FUNCTION_BLOCK FeedReactor3PsBasic (* Logica das 3 bombas de alimentacao (2 servico + 1 reserva) - mesmo funcionamento da Water Discharge *)
  (* Standard: 61499-2 *)
  (* Version 1.2, 10/7/2026, Claude/Hidryco, Schneider Electric, Rev3 - Velocidade das bombas sempre igual a saida do PID (1 ou 2 bombas); so muda para C2 na entrada/troca de bomba; sem fator 2, sem Cmin e sem capacidade teorica na falha do medidor | Rev2 - Setpoint do PID sempre igual ao setpoint do Nereda (removida a troca pela vazao medida com as bombas em C2) | Rev1 - Reescrito conforme a narrativa (cap. 2) com o mesmo funcionamento da Water Discharge (Rev13): Cmax/C2/C3/Cmin em % de velocidade; entrada da 2a com a bomba no Cmax pela velocidade real (narrativa); descida ate C2 confirmada pela velocidade real antes de partir a nova; T_C2 com as bombas em C2; reserva em falha parte na hora em C2; saida da 2a com protecao anti-ciclo; rodizio por horimetro; paradas por LL do buffer, pH/condutividade (L/H, retomada apos T_Restart) e vazao LL (T_FlowLL, retomada apos T_Restart); falha do medidor pela capacidade teorica; status para IHM *)
  PACKAGE SE.Nereda;
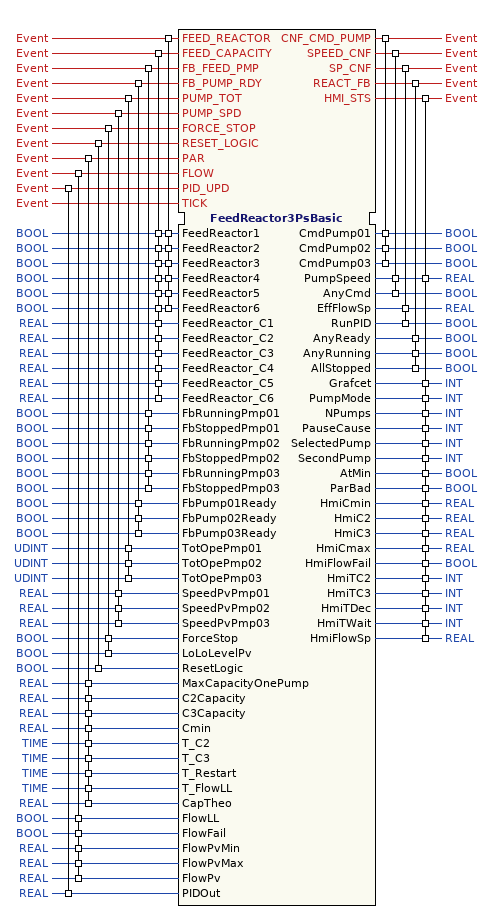
  EVENT_INPUT
    FEED_REACTOR WITH FeedReactor1, FeedReactor2, FeedReactor3, FeedReactor4, FeedReactor5, FeedReactor6; (* Pedido de alimentacao dos reatores (StartFeeding) *)
    FEED_CAPACITY WITH FeedReactor1, FeedReactor2, FeedReactor3, FeedReactor4, FeedReactor5, FeedReactor6, FeedReactor_C1, FeedReactor_C2, FeedReactor_C3, FeedReactor_C4, FeedReactor_C5, FeedReactor_C6; (* Setpoint de vazao dos reatores [m3/h] *)
    FB_FEED_PMP WITH FbRunningPmp01, FbStoppedPmp01, FbRunningPmp02, FbStoppedPmp02, FbRunningPmp03, FbStoppedPmp03;
    FB_PUMP_RDY WITH FbPump01Ready, FbPump02Ready, FbPump03Ready;
    PUMP_TOT WITH TotOpePmp01, TotOpePmp02, TotOpePmp03; (* Horimetro das bombas (rodizio) *)
    PUMP_SPD WITH SpeedPvPmp01, SpeedPvPmp02, SpeedPvPmp03; (* Velocidade real das bombas [%] *)
    FORCE_STOP WITH ForceStop, LoLoLevelPv; (* LL do buffer (40LT0001) e pH/condutividade fora da faixa (L/H) *)
    RESET_LOGIC WITH ResetLogic;
    PAR WITH MaxCapacityOnePump, C2Capacity, C3Capacity, Cmin, T_C2, T_C3, T_Restart, T_FlowLL, CapTheo; (* Parametros *)
    FLOW WITH FlowLL, FlowFail, FlowPvMin, FlowPvMax, FlowPv; (* Status e valor do 40FT0003 *)
    PID_UPD WITH PIDOut; (* Saida do PID *)
    TICK; (* Base de tempo 1 s *)
  END_EVENT
  EVENT_OUTPUT
    CNF_CMD_PUMP WITH CmdPump01, CmdPump02, CmdPump03; (* Comando das bombas *)
    SPEED_CNF WITH PumpSpeed, AnyCmd; (* Velocidade enviada a cada bomba em servico *)
    SP_CNF WITH EffFlowSp, RunPID; (* Setpoint efetivo e liberacao do PID *)
    REACT_FB WITH AnyReady, AnyRunning, AllStopped; (* Retorno das bombas para os reatores *)
    HMI_STS WITH Grafcet, PumpMode, NPumps, PauseCause, SelectedPump, SecondPump, PumpSpeed, AtMin, ParBad, HmiCmin, HmiC2, HmiC3, HmiCmax, HmiFlowFail, HmiTC2, HmiTC3, HmiTDec, HmiTWait, HmiFlowSp; (* Status para a IHM (a cada 1 s e na mudanca) *)
  END_EVENT
  VAR_INPUT
    FeedReactor1 : BOOL; (* StartFeeding do reator 1 (fase Feed em RUN e AV41101 aberta) *)
    FeedReactor2 : BOOL; (* StartFeeding do reator 2 (fase Feed em RUN e AV41101 aberta) *)
    FeedReactor3 : BOOL; (* StartFeeding do reator 3 (fase Feed em RUN e AV41101 aberta) *)
    FeedReactor4 : BOOL; (* StartFeeding do reator 4 (fase Feed em RUN e AV41101 aberta) *)
    FeedReactor5 : BOOL; (* StartFeeding do reator 5 (fase Feed em RUN e AV41101 aberta) *)
    FeedReactor6 : BOOL; (* StartFeeding do reator 6 (fase Feed em RUN e AV41101 aberta) *)
    FeedReactor_C1 : REAL; (* Setpoint de vazao do reator 1 [m3/h] *)
    FeedReactor_C2 : REAL; (* Setpoint de vazao do reator 2 [m3/h] *)
    FeedReactor_C3 : REAL; (* Setpoint de vazao do reator 3 [m3/h] *)
    FeedReactor_C4 : REAL; (* Setpoint de vazao do reator 4 [m3/h] *)
    FeedReactor_C5 : REAL; (* Setpoint de vazao do reator 5 [m3/h] *)
    FeedReactor_C6 : REAL; (* Setpoint de vazao do reator 6 [m3/h] *)
    FbRunningPmp01 : BOOL;
    FbStoppedPmp01 : BOOL;
    FbRunningPmp02 : BOOL;
    FbStoppedPmp02 : BOOL;
    FbRunningPmp03 : BOOL;
    FbStoppedPmp03 : BOOL;
    FbPump01Ready : BOOL;
    FbPump02Ready : BOOL;
    FbPump03Ready : BOOL;
    TotOpePmp01 : UDINT; (* Horimetro da bomba 1 *)
    TotOpePmp02 : UDINT; (* Horimetro da bomba 2 *)
    TotOpePmp03 : UDINT; (* Horimetro da bomba 3 *)
    SpeedPvPmp01 : REAL; (* Velocidade real da bomba 1 [%] *)
    SpeedPvPmp02 : REAL; (* Velocidade real da bomba 2 [%] *)
    SpeedPvPmp03 : REAL; (* Velocidade real da bomba 3 [%] *)
    ForceStop : BOOL; (* pH ou condutividade fora da faixa (alarmes L/H dos analisadores) *)
    LoLoLevelPv : BOOL; (* Nivel LL do buffer 40LT0001 *)
    ResetLogic : BOOL; (* Nao usado (compatibilidade) *)
    MaxCapacityOnePump : REAL; (* Cmax: velocidade de 1 bomba acima da qual entra a 2a [%] *)
    C2Capacity : REAL; (* C2: velocidade das bombas na entrada de uma nova bomba [%] *)
    C3Capacity : REAL; (* C3: velocidade das 2 bombas abaixo da qual sai 1 [%] *)
    Cmin : REAL; (* Nao atua desde a Rev3 (velocidade minima = OutMin do PID); so exibido na IHM *)
    T_C2 : TIME; (* Tempo com as bombas em C2 *)
    T_C3 : TIME; (* Tempo abaixo de C3 *)
    T_Restart : TIME; (* Tempo de espera para retomar a alimentacao (pH/condutividade/vazao LL) *)
    T_FlowLL : TIME; (* Vazao LL do 40FT0003 com bomba rodando por este tempo = para a alimentacao (0 = desabilitado) *)
    CapTheo : REAL; (* Nao usada desde a Rev3 (na falha do medidor as bombas seguem a saida do PID) *)
    FlowLL : BOOL; (* Alarme LL do 40FT0003 *)
    FlowFail : BOOL; (* Falha do 40FT0003 *)
    FlowPvMin : REAL; (* Inicio de faixa do 40FT0003 *)
    FlowPvMax : REAL; (* Fim de faixa do 40FT0003 *)
    FlowPv : REAL; (* Vazao medida 40FT0003 [m3/h] (nao usada desde a Rev2; mantida pela ligacao no FeedReactorLogic) *)
    PIDOut : REAL; (* Saida do PID = velocidade de cada bomba em servico [%] *)
  END_VAR
  VAR_OUTPUT
    CmdPump01 : BOOL;
    CmdPump02 : BOOL;
    CmdPump03 : BOOL;
    PumpSpeed : REAL; (* Velocidade enviada a cada bomba em servico [%] (= saida do PID; C2 na entrada/troca de bomba) *)
    AnyCmd : BOOL; (* Alguma bomba comandada *)
    EffFlowSp : REAL; (* Setpoint do PID [m3/h] = setpoint do Nereda (maior pedido entre os reatores alimentando) *)
    RunPID : BOOL; (* PID em automatico *)
    AnyReady : BOOL; (* Alguma bomba disponivel (Ready ou rodando) *)
    AnyRunning : BOOL; (* Alguma bomba rodando *)
    AllStopped : BOOL; (* Nenhuma bomba rodando *)
    Grafcet : INT; (* 0 sem pedido | 3 alimentando *)
    PumpMode : INT; (* 0=1 bomba 1=reduzindo p/ C2 2=nova bomba em C2 (T_C2) 3=duas no PID *)
    NPumps : INT; (* Bombas em servico rodando *)
    PauseCause : INT; (* 0 sem pausa | 1 nivel LL 40LT0001 | 2 pH/condutividade | 3 vazao LL 40FT0003 *)
    SelectedPump : INT; (* Bomba em servico ha mais tempo *)
    SecondPump : INT; (* Segunda bomba em servico *)
    AtMin : BOOL; (* Sempre FALSE desde a Rev3 (sem velocidade minima na logica) *)
    ParBad : BOOL; (* Parametros incoerentes (so aviso) *)
    HmiCmin : REAL;
    HmiC2 : REAL;
    HmiC3 : REAL;
    HmiCmax : REAL;
    HmiFlowFail : BOOL;
    HmiTC2 : INT; (* Tempo em C2 [s] *)
    HmiTC3 : INT; (* Tempo abaixo de C3 [s] *)
    HmiTDec : INT; (* Tempo descendo ate C2 [s] *)
    HmiTWait : INT; (* Tempo de espera para retomar [s] *)
    HmiFlowSp : REAL; (* Setpoint de vazao [m3/h] *)
  END_VAR
  VAR
    Paused : BOOL;
    FeedReq : BOOL;
    FlowSp : REAL;
    Dem : REAL;
    CminEff : REAL;
    C2Eff : REAL;
    SpdRaw : REAL;
    ParOk : BOOL;
    ExitCond : BOOL;
    Spare : BOOL;
    SpdAtC2 : BOOL;
    SpdUpC2 : BOOL;
    SpdAtMax : BOOL;
    NCmd : INT;
    NRun : INT;
    NWant : INT;
    PumpSel : INT;
    MinTot : UDINT;
    MinOrd : UDINT;
    Seq : UDINT;
    Ord1 : UDINT;
    Ord2 : UDINT;
    Ord3 : UDINT;
    Tacc : TIME;
    T3acc : TIME;
    Tdec : TIME;
    Tup : TIME;
    Trest : TIME;
    Tmax : TIME;
    Tll : TIME;
    TC2s : INT;
    TC3s : INT;
    TDecs : INT;
    TRests : INT;
    FromTick : BOOL;
    EdgeOut : BOOL;
    EdgeSpd : BOOL;
    EdgeSts : BOOL;
    EdgeCmd : BOOL;
    PrevSP : REAL;
    PrevRun : BOOL;
    PrevAR : BOOL;
    PrevARun : BOOL;
    PrevSpd : REAL;
    PrevAC : BOOL;
    PrevC1 : BOOL;
    PrevC2 : BOOL;
    PrevC3 : BOOL;
    PrevSPM : INT;
    PrevSNP : INT;
    PrevSPC : INT;
    PrevSGR : INT;
    PrevSAM : BOOL;
    PrevSPB : BOOL;
    TolC2 : REAL := 2.0; (* Parametro interno: tolerancia [%] para considerar a bomba em C2 *)
    T_DecMax : TIME := T#1m; (* Parametro interno: tempo maximo esperando a velocidade real chegar a C2 *)
    HystExit : REAL := 10.0; (* Parametro interno: margem [%] abaixo de Cmax para a bomba que fica apos a saida da 2a (anti-ciclo) *)
  END_VAR
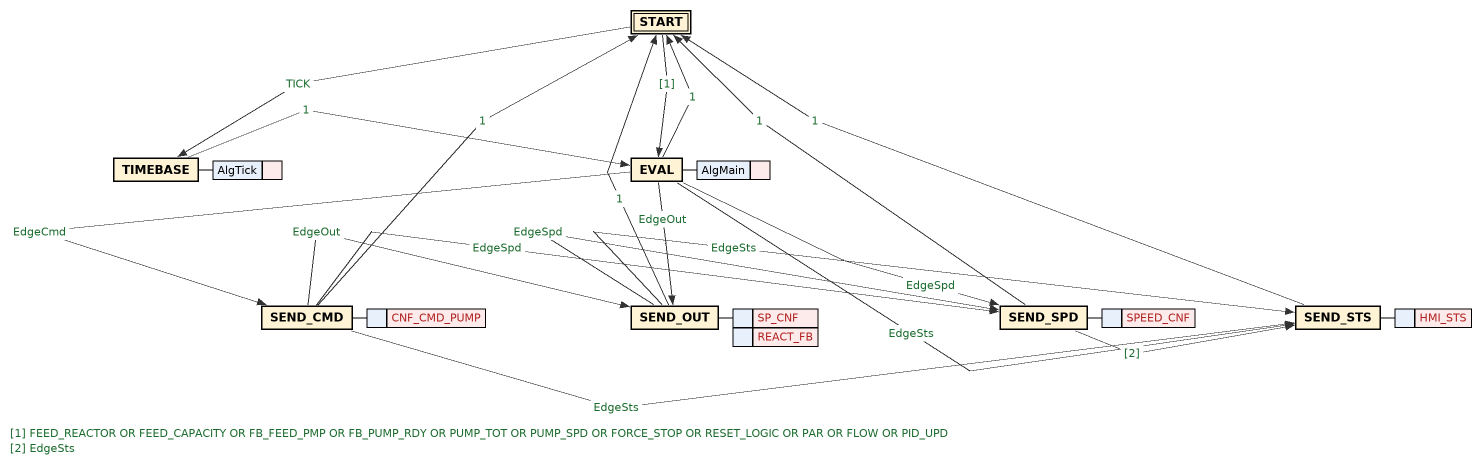
  EC_STATES
    START;
    TIMEBASE : AlgTick;
    EVAL : AlgMain;
    SEND_CMD : -> CNF_CMD_PUMP;
    SEND_OUT : -> SP_CNF, -> REACT_FB;
    SEND_SPD : -> SPEED_CNF;
    SEND_STS : -> HMI_STS;
  END_STATES
  EC_TRANSITIONS
    START TO TIMEBASE := TICK;
    START TO EVAL := FEED_REACTOR OR FEED_CAPACITY OR FB_FEED_PMP OR FB_PUMP_RDY OR PUMP_TOT OR PUMP_SPD OR FORCE_STOP OR RESET_LOGIC OR PAR OR FLOW OR PID_UPD;
    EVAL TO SEND_CMD := EdgeCmd;
    EVAL TO SEND_OUT := EdgeOut;
    EVAL TO SEND_SPD := EdgeSpd;
    EVAL TO SEND_STS := EdgeSts;
    EVAL TO START := 1;
    SEND_CMD TO SEND_OUT := EdgeOut;
    SEND_CMD TO SEND_SPD := EdgeSpd;
    SEND_CMD TO SEND_STS := EdgeSts;
    SEND_CMD TO START := 1;
    SEND_OUT TO SEND_SPD := EdgeSpd;
    SEND_OUT TO SEND_STS := EdgeSts;
    SEND_OUT TO START := 1;
    SEND_SPD TO SEND_STS := EdgeSts;
    SEND_SPD TO START := 1;
    SEND_STS TO START := 1;
    TIMEBASE TO EVAL := 1;
  END_TRANSITIONS
  ALGORITHM AlgMain IN ST: (* Logica das bombas de alimentacao *)
;
(* ============================================================
   FeedReactor3PsBasic Rev3 - bombas de alimentacao P4001/P4002/P4003 (2 servico + 1 reserva)
   Rev3: a velocidade das bombas e SEMPRE a saida do PID (1 ou 2 bombas). So muda para C2 na entrada/troca de bomba
         (modos 1 e 2). Sem fator 2 com uma bomba, sem velocidade minima (Cmin) e sem capacidade teorica na falha do medidor.
   Rev2: o setpoint do PID e sempre o setpoint do Nereda (removida a troca pela vazao medida com as bombas em C2).
   Narrativa cap. 2 (Influent feed) com o mesmo funcionamento da Water Discharge do Sludge Buffer.
   - Partida: StartFeeding de algum reator (fase Feed em RUN e AV41101 aberta). SP = maior pedido [m3/h].
   - Velocidade de cada bomba em servico = saida do PID [%]. Cmax / C2 / C3 em % de velocidade de UMA bomba.
     Limites de velocidade: OutMin/OutMax do proprio PID.
   - Entrada: velocidade REAL da bomba em operacao no Cmax -> a(s) em operacao descem ate C2 (velocidade REAL),
     a nova parte em C2, T_C2 com as duas com velocidade REAL em C2, depois PID. Sem liberacao por tempo.
   - Saida: velocidade REAL de todas as bombas em operacao abaixo de C3 por T_C3: sai a que partiu primeiro.
   - Falha de bomba com 2 em servico: reserva parte na hora, todas em C2, T_C2, depois PID.
   - Paradas: 1 nivel LL 40LT0001 (retoma ao sair o LL) | 2 pH/condutividade fora da faixa (retoma T_Restart apos voltar)
              3 vazao LL 40FT0003 por T_FlowLL com bomba rodando (retoma apos T_Restart)
   - Falha do 40FT0003 (40FT05): as bombas continuam seguindo a saida do PID (Rev3).
   PumpMode: 0 uma bomba | 1 reduzindo p/ C2 (nova parada) | 2 nova em C2 (T_C2) | 3 duas no PID
   ============================================================ *)

(* ---------- 1. Pedido de alimentacao e setpoint ---------- *)
FeedReq := FeedReactor1 OR FeedReactor2 OR FeedReactor3 OR FeedReactor4 OR FeedReactor5 OR FeedReactor6;
FlowSp := 0.0;
IF FeedReactor1 AND (FeedReactor_C1 > FlowSp) THEN
    FlowSp := FeedReactor_C1;
END_IF;
IF FeedReactor2 AND (FeedReactor_C2 > FlowSp) THEN
    FlowSp := FeedReactor_C2;
END_IF;
IF FeedReactor3 AND (FeedReactor_C3 > FlowSp) THEN
    FlowSp := FeedReactor_C3;
END_IF;
IF FeedReactor4 AND (FeedReactor_C4 > FlowSp) THEN
    FlowSp := FeedReactor_C4;
END_IF;
IF FeedReactor5 AND (FeedReactor_C5 > FlowSp) THEN
    FlowSp := FeedReactor_C5;
END_IF;
IF FeedReactor6 AND (FeedReactor_C6 > FlowSp) THEN
    FlowSp := FeedReactor_C6;
END_IF;
IF FeedReq THEN
    Grafcet := 3;
ELSE
    Grafcet := 0;
END_IF;

(* ---------- 2. Demanda e parametros ---------- *)
(* Rev3: a demanda e sempre a saida do PID (inclusive com o medidor em falha) *)
Dem := PIDOut;
IF Dem > 100.0 THEN
    Dem := 100.0;
END_IF;
IF Dem < 0.0 THEN
    Dem := 0.0;
END_IF;
CminEff := Cmin;
IF CminEff > 100.0 THEN
    CminEff := 100.0;
END_IF;
IF CminEff < 0.0 THEN
    CminEff := 0.0;
END_IF;
(* so Cmax e C2 sao indispensaveis; o resto apenas avisa (ParBad) - a protecao anti-ciclo esta embutida na saida *)
ParOk := (MaxCapacityOnePump > 0.0) AND (C2Capacity > 0.0);
(* Rev3: Cmin nao atua mais (velocidade minima = OutMin do PID); 2 x C3 >= Cmax continua causando ciclo de entrada/saida *)
ParBad := (MaxCapacityOnePump <= 0.0) OR (C2Capacity <= 0.0) OR ((2.0 * C3Capacity) >= MaxCapacityOnePump);
C2Eff := C2Capacity;
ExitCond := FALSE; (* calculado mais abaixo, so pela velocidade real das bombas *)

(* ---------- 3. Paradas da alimentacao (narrativa 2.2) ---------- *)
IF Grafcet = 3 THEN
    IF Paused THEN
        IF (PauseCause = 1) AND (NOT LoLoLevelPv) THEN
            Paused := FALSE;
            PauseCause := 0;
            Tll := T#0s;
        ELSIF (PauseCause >= 2) AND (NOT LoLoLevelPv) AND (NOT ForceStop) AND (Trest >= T_Restart) THEN
            Paused := FALSE;
            PauseCause := 0;
            Tll := T#0s;
        END_IF;
    END_IF;
    IF LoLoLevelPv THEN
        Paused := TRUE;
        PauseCause := 1;
        Trest := T#0s;
        TRests := 0;
    ELSIF ForceStop THEN
        Paused := TRUE;
        PauseCause := 2;
        Trest := T#0s;
        TRests := 0;
    ELSIF (NOT Paused) AND (T_FlowLL > T#0s) AND (Tll >= T_FlowLL) THEN
        Paused := TRUE;
        PauseCause := 3;
        Trest := T#0s;
        TRests := 0;
        Tll := T#0s;
    END_IF;
END_IF;

(* ---------- 4. Bombas ---------- *)
IF (Grafcet = 3) AND Paused THEN
    CmdPump01 := FALSE;
    CmdPump02 := FALSE;
    CmdPump03 := FALSE;
    PumpMode := 0;
    Tacc := T#0s;
    TC2s := 0;
    T3acc := T#0s;
    TC3s := 0;
    NCmd := 0;
    NRun := 0;
    EffFlowSp := FlowSp;
    PumpSpeed := 0.0;
    AtMin := FALSE;
ELSIF Grafcet = 3 THEN
    (* 4.1 bomba sai de servico somente se nao estiver Ready (modo programa) NEM Running *)
    IF CmdPump01 AND NOT FbPump01Ready AND NOT FbRunningPmp01 THEN
        CmdPump01 := FALSE;
    END_IF;
    IF CmdPump02 AND NOT FbPump02Ready AND NOT FbRunningPmp02 THEN
        CmdPump02 := FALSE;
    END_IF;
    IF CmdPump03 AND NOT FbPump03Ready AND NOT FbRunningPmp03 THEN
        CmdPump03 := FALSE;
    END_IF;
    NCmd := 0;
    IF CmdPump01 THEN
        NCmd := NCmd + 1;
    END_IF;
    IF CmdPump02 THEN
        NCmd := NCmd + 1;
    END_IF;
    IF CmdPump03 THEN
        NCmd := NCmd + 1;
    END_IF;
    NRun := 0;
    IF CmdPump01 AND FbRunningPmp01 THEN
        NRun := NRun + 1;
    END_IF;
    IF CmdPump02 AND FbRunningPmp02 THEN
        NRun := NRun + 1;
    END_IF;
    IF CmdPump03 AND FbRunningPmp03 THEN
        NRun := NRun + 1;
    END_IF;
    Spare := (FbPump01Ready AND NOT CmdPump01) OR (FbPump02Ready AND NOT CmdPump02) OR (FbPump03Ready AND NOT CmdPump03);
    (* bombas em operacao ja desceram ate C2 (velocidade real) *)
    SpdAtC2 := TRUE;
    IF CmdPump01 AND FbRunningPmp01 AND (SpeedPvPmp01 > (C2Eff + TolC2)) THEN
        SpdAtC2 := FALSE;
    END_IF;
    IF CmdPump02 AND FbRunningPmp02 AND (SpeedPvPmp02 > (C2Eff + TolC2)) THEN
        SpdAtC2 := FALSE;
    END_IF;
    IF CmdPump03 AND FbRunningPmp03 AND (SpeedPvPmp03 > (C2Eff + TolC2)) THEN
        SpdAtC2 := FALSE;
    END_IF;
    (* bomba em operacao com velocidade real ja no Cmax *)
    SpdAtMax := FALSE;
    IF CmdPump01 AND FbRunningPmp01 AND (SpeedPvPmp01 >= (MaxCapacityOnePump - TolC2)) THEN
        SpdAtMax := TRUE;
    END_IF;
    IF CmdPump02 AND FbRunningPmp02 AND (SpeedPvPmp02 >= (MaxCapacityOnePump - TolC2)) THEN
        SpdAtMax := TRUE;
    END_IF;
    IF CmdPump03 AND FbRunningPmp03 AND (SpeedPvPmp03 >= (MaxCapacityOnePump - TolC2)) THEN
        SpdAtMax := TRUE;
    END_IF;
    (* bombas em operacao com velocidade real ja em C2 (subida da que entrou) *)
    SpdUpC2 := TRUE;
    IF CmdPump01 AND FbRunningPmp01 AND (SpeedPvPmp01 < (C2Eff - TolC2)) THEN
        SpdUpC2 := FALSE;
    END_IF;
    IF CmdPump02 AND FbRunningPmp02 AND (SpeedPvPmp02 < (C2Eff - TolC2)) THEN
        SpdUpC2 := FALSE;
    END_IF;
    IF CmdPump03 AND FbRunningPmp03 AND (SpeedPvPmp03 < (C2Eff - TolC2)) THEN
        SpdUpC2 := FALSE;
    END_IF;
    (* saida de uma bomba: velocidade real de TODAS as bombas em operacao abaixo de C3 (sem usar a saida do PID) *)
    ExitCond := NRun >= 2;
    IF CmdPump01 AND FbRunningPmp01 AND (SpeedPvPmp01 >= C3Capacity) THEN
        ExitCond := FALSE;
    END_IF;
    IF CmdPump02 AND FbRunningPmp02 AND (SpeedPvPmp02 >= C3Capacity) THEN
        ExitCond := FALSE;
    END_IF;
    IF CmdPump03 AND FbRunningPmp03 AND (SpeedPvPmp03 >= C3Capacity) THEN
        ExitCond := FALSE;
    END_IF;
    (* 4.1b com 2 bombas (modo 2/3) uma saiu de servico: a reserva parte NA HORA, todas em C2, T_C2, depois PID *)
    IF ParOk AND (PumpMode >= 2) AND (NCmd < 2) THEN
        IF Spare AND (NCmd >= 1) THEN
            PumpMode := 2;
            Tacc := T#0s;
            TC2s := 0;
            Tup := T#0s;
        ELSE
            PumpMode := 0;
        END_IF;
    END_IF;

    (* 4.2 numero de bombas *)
    IF NOT ParOk THEN
        PumpMode := 0;
    ELSIF PumpMode = 0 THEN
        (* entra a 2a bomba somente quando a velocidade REAL da bomba em operacao chega ao Cmax *)
        IF Spare AND (NRun >= 1) AND SpdAtMax THEN
            PumpMode := 1;
            Tdec := T#0s;
            TDecs := 0;
        END_IF;
    ELSIF PumpMode = 1 THEN
        (* a nova so parte depois que a velocidade REAL da(s) bomba(s) em operacao desceu ate C2 *)
        IF (NOT Spare) OR (NCmd = 0) THEN
            PumpMode := 0;
        ELSIF SpdAtC2 THEN
            PumpMode := 2;
            Tacc := T#0s;
            TC2s := 0;
            Tup := T#0s;
        END_IF;
    ELSIF PumpMode = 2 THEN
        (* T_C2 conta com as duas rodando e com velocidade REAL em C2 *)
        IF (NRun >= 2) AND (Tacc >= T_C2) THEN
            PumpMode := 3;
            T3acc := T#0s;
            TC3s := 0;
        END_IF;
    ELSIF PumpMode = 3 THEN
        (* saida: velocidade REAL das bombas abaixo de C3 por T_C3 *)
        IF ExitCond AND (T3acc >= T_C3) THEN
            PumpMode := 0;
            T3acc := T#0s;
            TC3s := 0;
        END_IF;
    END_IF;
    IF PumpMode >= 2 THEN
        NWant := 2;
    ELSE
        NWant := 1;
    END_IF;

    (* 4.3 entra bomba disponivel de menor horimetro (rodizio) - ate 2 vezes *)
    IF NCmd < NWant THEN
        PumpSel := 0;
        IF FbPump01Ready AND NOT CmdPump01 THEN
            PumpSel := 1;
            MinTot := TotOpePmp01;
        END_IF;
        IF FbPump02Ready AND NOT CmdPump02 THEN
            IF (PumpSel = 0) OR (TotOpePmp02 < MinTot) THEN
                PumpSel := 2;
                MinTot := TotOpePmp02;
            END_IF;
        END_IF;
        IF FbPump03Ready AND NOT CmdPump03 THEN
            IF (PumpSel = 0) OR (TotOpePmp03 < MinTot) THEN
                PumpSel := 3;
                MinTot := TotOpePmp03;
            END_IF;
        END_IF;
        IF PumpSel = 1 THEN
            CmdPump01 := TRUE;
            Seq := Seq + 1;
            Ord1 := Seq;
            NCmd := NCmd + 1;
        ELSIF PumpSel = 2 THEN
            CmdPump02 := TRUE;
            Seq := Seq + 1;
            Ord2 := Seq;
            NCmd := NCmd + 1;
        ELSIF PumpSel = 3 THEN
            CmdPump03 := TRUE;
            Seq := Seq + 1;
            Ord3 := Seq;
            NCmd := NCmd + 1;
        END_IF;
    END_IF;
    IF NCmd < NWant THEN
        PumpSel := 0;
        IF FbPump01Ready AND NOT CmdPump01 THEN
            PumpSel := 1;
            MinTot := TotOpePmp01;
        END_IF;
        IF FbPump02Ready AND NOT CmdPump02 THEN
            IF (PumpSel = 0) OR (TotOpePmp02 < MinTot) THEN
                PumpSel := 2;
                MinTot := TotOpePmp02;
            END_IF;
        END_IF;
        IF FbPump03Ready AND NOT CmdPump03 THEN
            IF (PumpSel = 0) OR (TotOpePmp03 < MinTot) THEN
                PumpSel := 3;
                MinTot := TotOpePmp03;
            END_IF;
        END_IF;
        IF PumpSel = 1 THEN
            CmdPump01 := TRUE;
            Seq := Seq + 1;
            Ord1 := Seq;
            NCmd := NCmd + 1;
        ELSIF PumpSel = 2 THEN
            CmdPump02 := TRUE;
            Seq := Seq + 1;
            Ord2 := Seq;
            NCmd := NCmd + 1;
        ELSIF PumpSel = 3 THEN
            CmdPump03 := TRUE;
            Seq := Seq + 1;
            Ord3 := Seq;
            NCmd := NCmd + 1;
        END_IF;
    END_IF;

    (* 4.4 excedente: sai a bomba em operacao ha mais tempo (menor ordem de partida) *)
    IF NCmd > NWant THEN
        PumpSel := 0;
        IF CmdPump01 THEN
            PumpSel := 1;
            MinOrd := Ord1;
        END_IF;
        IF CmdPump02 THEN
            IF (PumpSel = 0) OR (Ord2 < MinOrd) THEN
                PumpSel := 2;
                MinOrd := Ord2;
            END_IF;
        END_IF;
        IF CmdPump03 THEN
            IF (PumpSel = 0) OR (Ord3 < MinOrd) THEN
                PumpSel := 3;
                MinOrd := Ord3;
            END_IF;
        END_IF;
        IF PumpSel = 1 THEN
            CmdPump01 := FALSE;
        ELSIF PumpSel = 2 THEN
            CmdPump02 := FALSE;
        ELSIF PumpSel = 3 THEN
            CmdPump03 := FALSE;
        END_IF;
        NCmd := NCmd - 1;
    END_IF;

    (* 4.5 sem bomba para a 2a posicao: volta a operar com uma *)
    IF (PumpMode >= 2) AND (NCmd < 2) THEN
        PumpMode := 0;
    END_IF;

    (* 4.6 setpoint do PID e velocidade das bombas *)
    (* setpoint do PID = setpoint do Nereda (maior pedido), sempre - nunca trocado pela vazao medida (Rev2) *)
    EffFlowSp := FlowSp;
    (* Rev3: velocidade de cada bomba = saida do PID; a unica sobreposicao e C2 na entrada/troca de bomba (modos 1 e 2) *)
    IF (PumpMode = 1) OR (PumpMode = 2) THEN
        SpdRaw := C2Eff;
    ELSE
        SpdRaw := Dem;
    END_IF;
    IF SpdRaw > 100.0 THEN
        SpdRaw := 100.0;
    END_IF;
    IF SpdRaw < 0.0 THEN
        SpdRaw := 0.0;
    END_IF;
    AtMin := FALSE; (* Rev3: sem velocidade minima na logica *)
    PumpSpeed := SpdRaw;
ELSE
    (* sem pedido de alimentacao *)
    CmdPump01 := FALSE;
    CmdPump02 := FALSE;
    CmdPump03 := FALSE;
    PumpMode := 0;
    Tacc := T#0s;
    TC2s := 0;
    T3acc := T#0s;
    TC3s := 0;
    NCmd := 0;
    NRun := 0;
    EffFlowSp := FlowSp;
    PumpSpeed := 0.0;
    AtMin := FALSE;
    Paused := FALSE;
    PauseCause := 0;
    Trest := T#0s;
    TRests := 0;
    Tll := T#0s;
END_IF;

(* ---------- 5. Saidas ---------- *)
AnyCmd := CmdPump01 OR CmdPump02 OR CmdPump03;
RunPID := (Grafcet = 3) AND (NOT Paused) AND AnyCmd;
AnyReady := FbPump01Ready OR FbRunningPmp01 OR FbPump02Ready OR FbRunningPmp02 OR FbPump03Ready OR FbRunningPmp03;
AnyRunning := FbRunningPmp01 OR FbRunningPmp02 OR FbRunningPmp03;
AllStopped := NOT AnyRunning;
NPumps := NRun;
SelectedPump := 0;
SecondPump := 0;
MinOrd := 0;
IF CmdPump01 THEN
    SelectedPump := 1;
    MinOrd := Ord1;
END_IF;
IF CmdPump02 THEN
    IF (SelectedPump = 0) OR (Ord2 < MinOrd) THEN
        SecondPump := SelectedPump;
        SelectedPump := 2;
        MinOrd := Ord2;
    ELSE
        SecondPump := 2;
    END_IF;
END_IF;
IF CmdPump03 THEN
    IF (SelectedPump = 0) OR (Ord3 < MinOrd) THEN
        SecondPump := SelectedPump;
        SelectedPump := 3;
        MinOrd := Ord3;
    ELSE
        SecondPump := 3;
    END_IF;
END_IF;

(* ---------- 6. Eventos de saida somente na mudanca ---------- *)
EdgeCmd := (CmdPump01 <> PrevC1) OR (CmdPump02 <> PrevC2) OR (CmdPump03 <> PrevC3);
PrevC1 := CmdPump01;
PrevC2 := CmdPump02;
PrevC3 := CmdPump03;
EdgeOut := (EffFlowSp <> PrevSP) OR (RunPID <> PrevRun) OR (AnyReady <> PrevAR) OR (AnyRunning <> PrevARun);
PrevSP := EffFlowSp;
PrevRun := RunPID;
PrevAR := AnyReady;
PrevARun := AnyRunning;
EdgeSpd := (PumpSpeed <> PrevSpd) OR (AnyCmd <> PrevAC);
PrevSpd := PumpSpeed;
PrevAC := AnyCmd;

(* ---------- 7. Status para a IHM: a cada 1 s (TICK) e quando o estado muda ---------- *)
HmiCmin := CminEff;
HmiC2 := C2Eff;
HmiC3 := C3Capacity;
HmiCmax := MaxCapacityOnePump;
HmiFlowFail := FlowFail;
HmiTC2 := TC2s;
HmiTC3 := TC3s;
HmiTDec := TDecs;
HmiTWait := TRests;
HmiFlowSp := FlowSp;
EdgeSts := FromTick OR (PumpMode <> PrevSPM) OR (NPumps <> PrevSNP) OR (PauseCause <> PrevSPC) OR (Grafcet <> PrevSGR) OR (AtMin <> PrevSAM) OR (ParBad <> PrevSPB);
FromTick := FALSE;
PrevSPM := PumpMode;
PrevSNP := NPumps;
PrevSPC := PauseCause;
PrevSGR := Grafcet;
PrevSAM := AtMin;
PrevSPB := ParBad;
  END_ALGORITHM
  ALGORITHM AlgTick IN ST: (* Base de tempo 1 s *)
;
(* Base de tempo 1 s (E_CYCLE externo) *)
FromTick := TRUE;
IF PumpMode = 2 THEN
    Tup := Tup + T#1s;
ELSE
    Tup := T#0s;
END_IF;
(* T_C2: as duas rodando e com velocidade REAL em C2 *)
IF (PumpMode = 2) AND (NRun >= 2) AND SpdUpC2 THEN
    Tacc := Tacc + T#1s;
    TC2s := TC2s + 1;
END_IF;
(* demanda acima do Cmax com 1 bomba (limite quando a velocidade real nao confirma o Cmax) *)
IF (PumpMode = 0) AND (NRun >= 1) AND (Dem > MaxCapacityOnePump) THEN
    Tmax := Tmax + T#1s;
ELSE
    Tmax := T#0s;
END_IF;
(* tempo de descida ate C2 antes de partir a nova bomba *)
IF PumpMode = 1 THEN
    Tdec := Tdec + T#1s;
    TDecs := TDecs + 1;
ELSE
    Tdec := T#0s;
    TDecs := 0;
END_IF;
(* duas bombas com a condicao de saida *)
IF (PumpMode = 3) AND (NRun >= 2) AND ExitCond THEN
    T3acc := T3acc + T#1s;
    TC3s := TC3s + 1;
ELSE
    T3acc := T#0s;
    TC3s := 0;
END_IF;
(* espera para retomar: conta so com as causas ja normalizadas *)
IF (Grafcet = 3) AND Paused AND (NOT LoLoLevelPv) AND (NOT ForceStop) THEN
    Trest := Trest + T#1s;
    TRests := TRests + 1;
ELSE
    Trest := T#0s;
    TRests := 0;
END_IF;
(* vazao LL com bomba rodando *)
IF (Grafcet = 3) AND (NOT Paused) AND (NRun >= 1) AND FlowLL AND (NOT FlowFail) THEN
    Tll := Tll + T#1s;
ELSE
    Tll := T#0s;
END_IF;
  END_ALGORITHM
END_FUNCTION_BLOCK
